// TIA Portal V17 export
// export: Created 2023-12-22T15:07:59.6202933Z, ExportSetting WithDefaults, DisplayName Totally Integrated Automation Portal, DisplayVersion V17, DisplayName TIA Portal Openness, DisplayVersion V17, DisplayName TIA Portal Version Control Interface, DisplayVersion V17, DisplayName STEP 7 Professional, DisplayVersion V17, DisplayName STEP 7 Safety, DisplayVersion V17, DisplayName WinCC Advanced, DisplayVersion V17
FUNCTION_BLOCK "PS_StartUp"   // FB13, LAD
{ S7_Optimized_Access := 'FALSE' }
VERSION : 0.1
// stored: AutoNumber false, IsIECCheckEnabled false, SetENOAutomatically false, UDAEnableTagReadback false
   VAR_INPUT
      PE : Real;
      LE_Target : Real;
      LE_Source : Real;
   END_VAR
   VAR_IN_OUT
      REQ : Int;
      Hz : Real;
   END_VAR
   VAR DB_SPECIFIC
      Start : Bool;   // Запуск системы
      Ready : Bool;   // Линия заполнена
      "Step" : Int;
      Warning : Word;
      PE_Point : Real;   // Давление на момент выхода плавный разгон
      PE_Delta : Real := 0.05;   // Допустимое отклонение
      PE_Min : Real;
      LE_Target_Point : Real;
      LE_Target_Delta : Real;
      LE_Target_Min : Real;
      LE_Source_Point : Real;
      LE_Source_Delta : Real;
      LE_Source_Min : Real;
      xSP : Array[0..5] of Struct
         Use { S7_SetPoint := 'True'} : Bool;
         REQ { S7_SetPoint := 'True'} : Int;
         Hz { S7_SetPoint := 'True'} : Real;
         PE { S7_SetPoint := 'True'} : Real;
         PE_Delta : Real;
      END_STRUCT;
   END_VAR
   VAR
      xTime { S7_SetPoint := 'True'} : Array[0..5] of "Time_M";
   END_VAR
   VAR_TEMP   // added for the SCL form of the ladder/FBD networks
      _w1 : Bool;
      _w2 : Bool;
      _w3 : Bool;
      _w4 : Bool;
      _w5 : Bool;
   END_VAR
BEGIN

REGION Network 1: 0 - Первичное заполнение труб
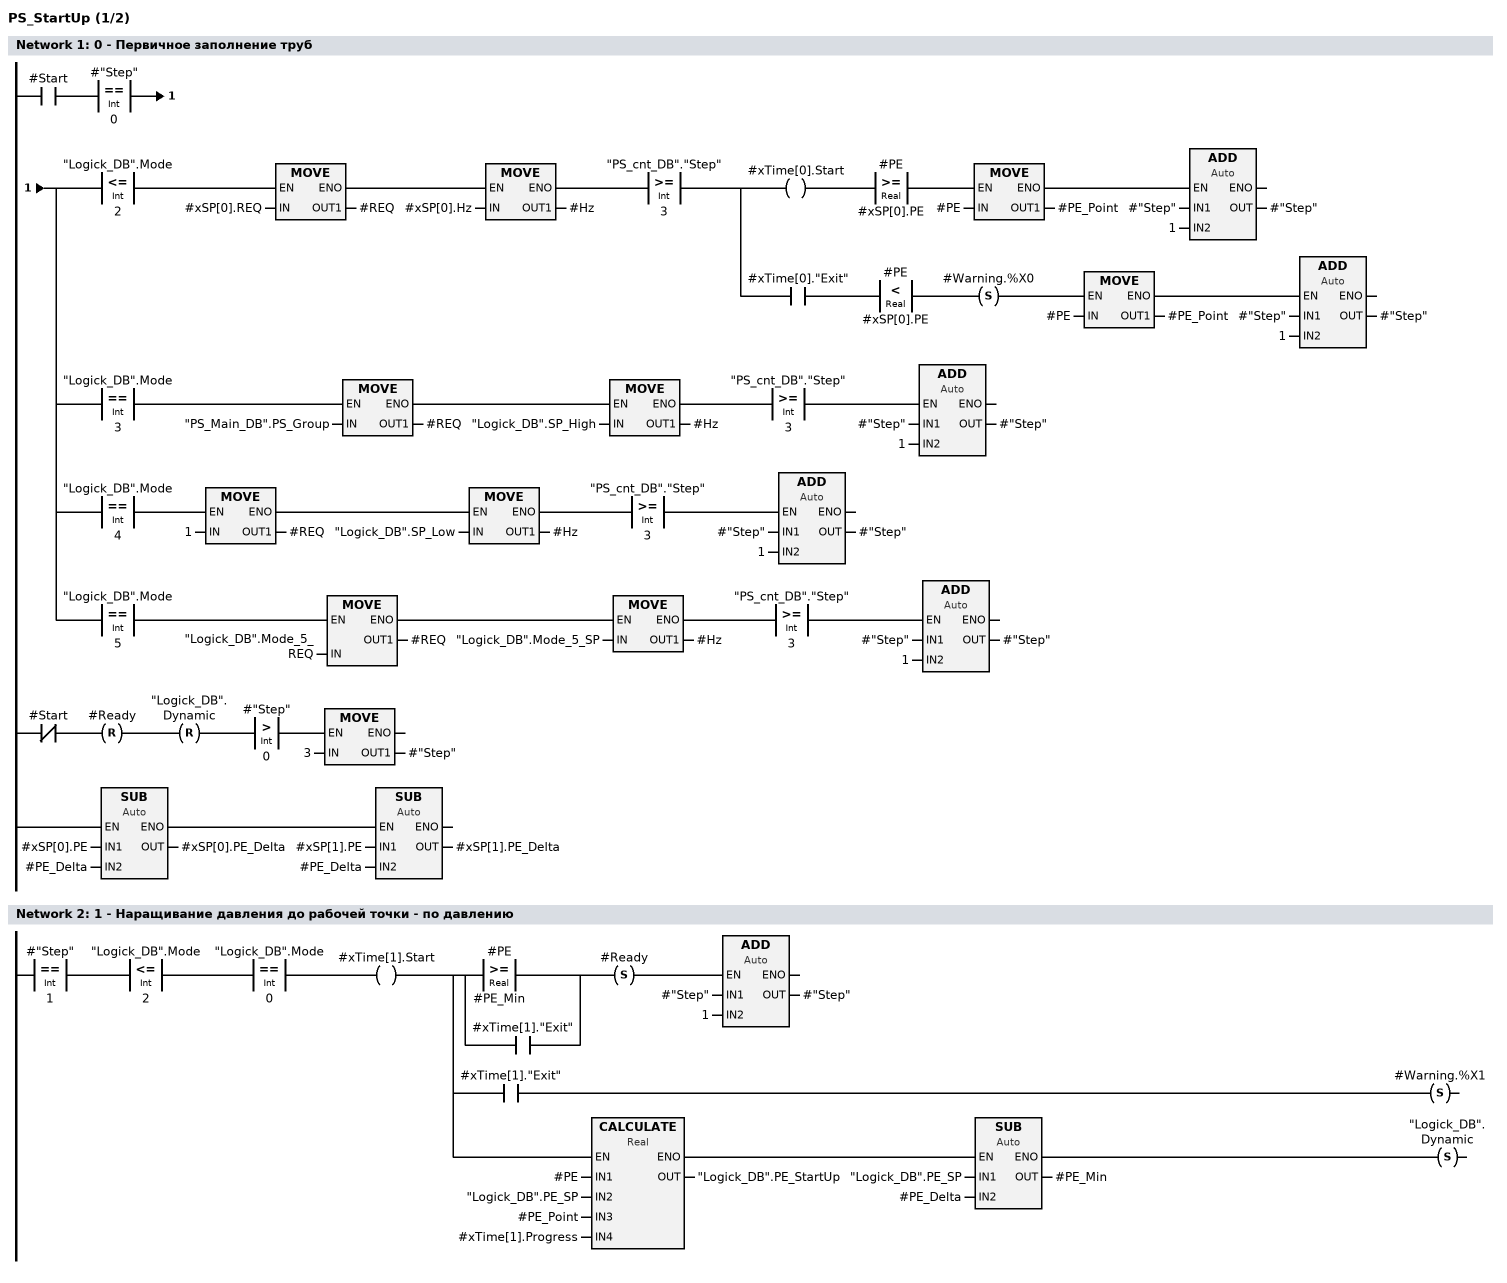
   RUNG wire#powerrail
      Contact( #Start )
      { S7_Templates := "SrcType := Int" } EQ_Contact(in1 := #"Step", in2 := 0)
      wire#w1
      { S7_Templates := "SrcType := Int" } LE_Contact(in1 := "Logick_DB".Mode, in2 := 2)
      Move(in := #xSP[0].REQ, out1 => #REQ)
      Move(in := #xSP[0].Hz, out1 => #Hz)
      { S7_Templates := "SrcType := Int" } GE_Contact(in1 := "PS_cnt_DB"."Step", in2 := 3)
      wire#w2
      Coil( #xTime[0].Start )
      { S7_Templates := "SrcType := Real" } GE_Contact(in1 := #PE, in2 := #xSP[0].PE)
      Move(in := #PE, out1 => #PE_Point)
      Add(in1 := #"Step", in2 := 1, out => #"Step")
   END_RUNG
   RUNG wire#w2
      Contact( #xTime[0]."Exit" )
      { S7_Templates := "SrcType := Real" } LT_Contact(in1 := #PE, in2 := #xSP[0].PE)
      S_Coil( #Warning.%X0 )
      Move(in := #PE, out1 => #PE_Point)
      Add(in1 := #"Step", in2 := 1, out => #"Step")
   END_RUNG
   RUNG wire#w1
      { S7_Templates := "SrcType := Int" } EQ_Contact(in1 := "Logick_DB".Mode, in2 := 3)
      Move(in := "PS_Main_DB".PS_Group, out1 => #REQ)
      Move(in := "Logick_DB".SP_High, out1 => #Hz)
      { S7_Templates := "SrcType := Int" } GE_Contact(in1 := "PS_cnt_DB"."Step", in2 := 3)
      Add(in1 := #"Step", in2 := 1, out => #"Step")
   END_RUNG
   RUNG wire#w1
      { S7_Templates := "SrcType := Int" } EQ_Contact(in1 := "Logick_DB".Mode, in2 := 4)
      Move(in := 1, out1 => #REQ)
      Move(in := "Logick_DB".SP_Low, out1 => #Hz)
      { S7_Templates := "SrcType := Int" } GE_Contact(in1 := "PS_cnt_DB"."Step", in2 := 3)
      Add(in1 := #"Step", in2 := 1, out => #"Step")
   END_RUNG
   RUNG wire#w1
      { S7_Templates := "SrcType := Int" } EQ_Contact(in1 := "Logick_DB".Mode, in2 := 5)
      Move(in := "Logick_DB".Mode_5_REQ, out1 => #REQ)
      Move(in := "Logick_DB".Mode_5_SP, out1 => #Hz)
      { S7_Templates := "SrcType := Int" } GE_Contact(in1 := "PS_cnt_DB"."Step", in2 := 3)
      Add(in1 := #"Step", in2 := 1, out => #"Step")
   END_RUNG
   RUNG wire#powerrail
      I_Contact( #Start )
      R_Coil( #Ready )
      R_Coil( "Logick_DB".Dynamic )
      { S7_Templates := "SrcType := Int" } GT_Contact(in1 := #"Step", in2 := 0)
      Move(in := 3, out1 => #"Step")
   END_RUNG
   RUNG wire#powerrail
      Sub(in1 := #xSP[0].PE, in2 := #PE_Delta, out => #xSP[0].PE_Delta)
      Sub(in1 := #xSP[1].PE, in2 := #PE_Delta, out => #xSP[1].PE_Delta)
   END_RUNG
   // the same network as SCL:
   #_w1 := #Start AND (#"Step" = 0);
   #_w2 := #_w1 AND ("Logick_DB".Mode <= 2);
   IF #_w2 THEN
       #REQ := #xSP[0].REQ;
       #Hz := #xSP[0].Hz;
   END_IF;
   #xTime[0].Start := #_w2 AND ("PS_cnt_DB"."Step" >= 3);
   IF #_w2 AND ("PS_cnt_DB"."Step" >= 3) AND (#PE >= #xSP[0].PE) THEN
       #PE_Point := #PE;
       #"Step" := #"Step" + 1;
   END_IF;
   IF #_w2 AND ("PS_cnt_DB"."Step" >= 3) AND #xTime[0]."Exit" AND (#PE < #xSP[0].PE) THEN
       #Warning.%X0 := TRUE;
       #PE_Point := #PE;
       #"Step" := #"Step" + 1;
   END_IF;
   #_w3 := #_w1 AND ("Logick_DB".Mode = 3);
   IF #_w3 THEN
       #REQ := "PS_Main_DB".PS_Group;
       #Hz := "Logick_DB".SP_High;
   END_IF;
   IF #_w3 AND ("PS_cnt_DB"."Step" >= 3) THEN #"Step" := #"Step" + 1; END_IF;
   #_w4 := #_w1 AND ("Logick_DB".Mode = 4);
   IF #_w4 THEN
       #REQ := 1;
       #Hz := "Logick_DB".SP_Low;
   END_IF;
   IF #_w4 AND ("PS_cnt_DB"."Step" >= 3) THEN #"Step" := #"Step" + 1; END_IF;
   #_w5 := #_w1 AND ("Logick_DB".Mode = 5);
   IF #_w5 THEN
       #REQ := "Logick_DB".Mode_5_REQ;
       #Hz := "Logick_DB".Mode_5_SP;
   END_IF;
   IF #_w5 AND ("PS_cnt_DB"."Step" >= 3) THEN #"Step" := #"Step" + 1; END_IF;
   IF NOT #Start THEN
       #Ready := FALSE;
       "Logick_DB".Dynamic := FALSE;
   END_IF;
   IF NOT #Start AND (#"Step" > 0) THEN #"Step" := 3; END_IF;
   #xSP[0].PE_Delta := #xSP[0].PE - #PE_Delta;
   #xSP[1].PE_Delta := #xSP[1].PE - #PE_Delta;
END_REGION

REGION Network 2: 1 - Наращивание давления до рабочей точки - по давлению
   RUNG wire#powerrail
      { S7_Templates := "SrcType := Int" } EQ_Contact(in1 := #"Step", in2 := 1)
      { S7_Templates := "SrcType := Int" } LE_Contact(in1 := "Logick_DB".Mode, in2 := 2)
      { S7_Templates := "SrcType := Int" } EQ_Contact(in1 := "Logick_DB".Mode, in2 := 0)
      Coil( #xTime[1].Start )
      wire#w1
      { S7_Templates := "SrcType := Real" } GE_Contact(in1 := #PE, in2 := #PE_Min)
      wire#w2
      S_Coil( #Ready )
      Add(in1 := #"Step", in2 := 1, out => #"Step")
   END_RUNG
   RUNG wire#w1
      Contact( #xTime[1]."Exit" )
   END_RUNG wire#w2
   RUNG wire#w1
      Contact( #xTime[1]."Exit" )
      S_Coil( #Warning.%X1 )
   END_RUNG
   RUNG wire#w1
      { S7_Templates := "SrcType := Real"; S7_Expression := "IN1 + (IN2 - IN3) * IN4" } Calculate(in1 := #PE, in2 := "Logick_DB".PE_SP, in3 := #PE_Point, in4 := #xTime[1].Progress, out => "Logick_DB".PE_StartUp)
      Sub(in1 := "Logick_DB".PE_SP, in2 := #PE_Delta, out => #PE_Min)
      S_Coil( "Logick_DB".Dynamic )
   END_RUNG
   // the same network as SCL:
   #xTime[1].Start := (#"Step" = 1) AND ("Logick_DB".Mode <= 2) AND ("Logick_DB".Mode = 0);
   #_w1 := (#"Step" = 1) AND ("Logick_DB".Mode <= 2) AND ("Logick_DB".Mode = 0);
   IF #_w1 AND ((#PE >= #PE_Min) OR #xTime[1]."Exit") THEN
       #Ready := TRUE;
       #"Step" := #"Step" + 1;
   END_IF;
   IF #_w1 AND #xTime[1]."Exit" THEN #Warning.%X1 := TRUE; END_IF;
   IF #_w1 THEN
       "Logick_DB".PE_StartUp := #PE + ("Logick_DB".PE_SP - #PE_Point) * #xTime[1].Progress;
       #PE_Min := "Logick_DB".PE_SP - #PE_Delta;
       "Logick_DB".Dynamic := TRUE;
   END_IF;
END_REGION

REGION Network 3: 1 - Наращивание давления до рабочей точки - по уровню в РЧВ
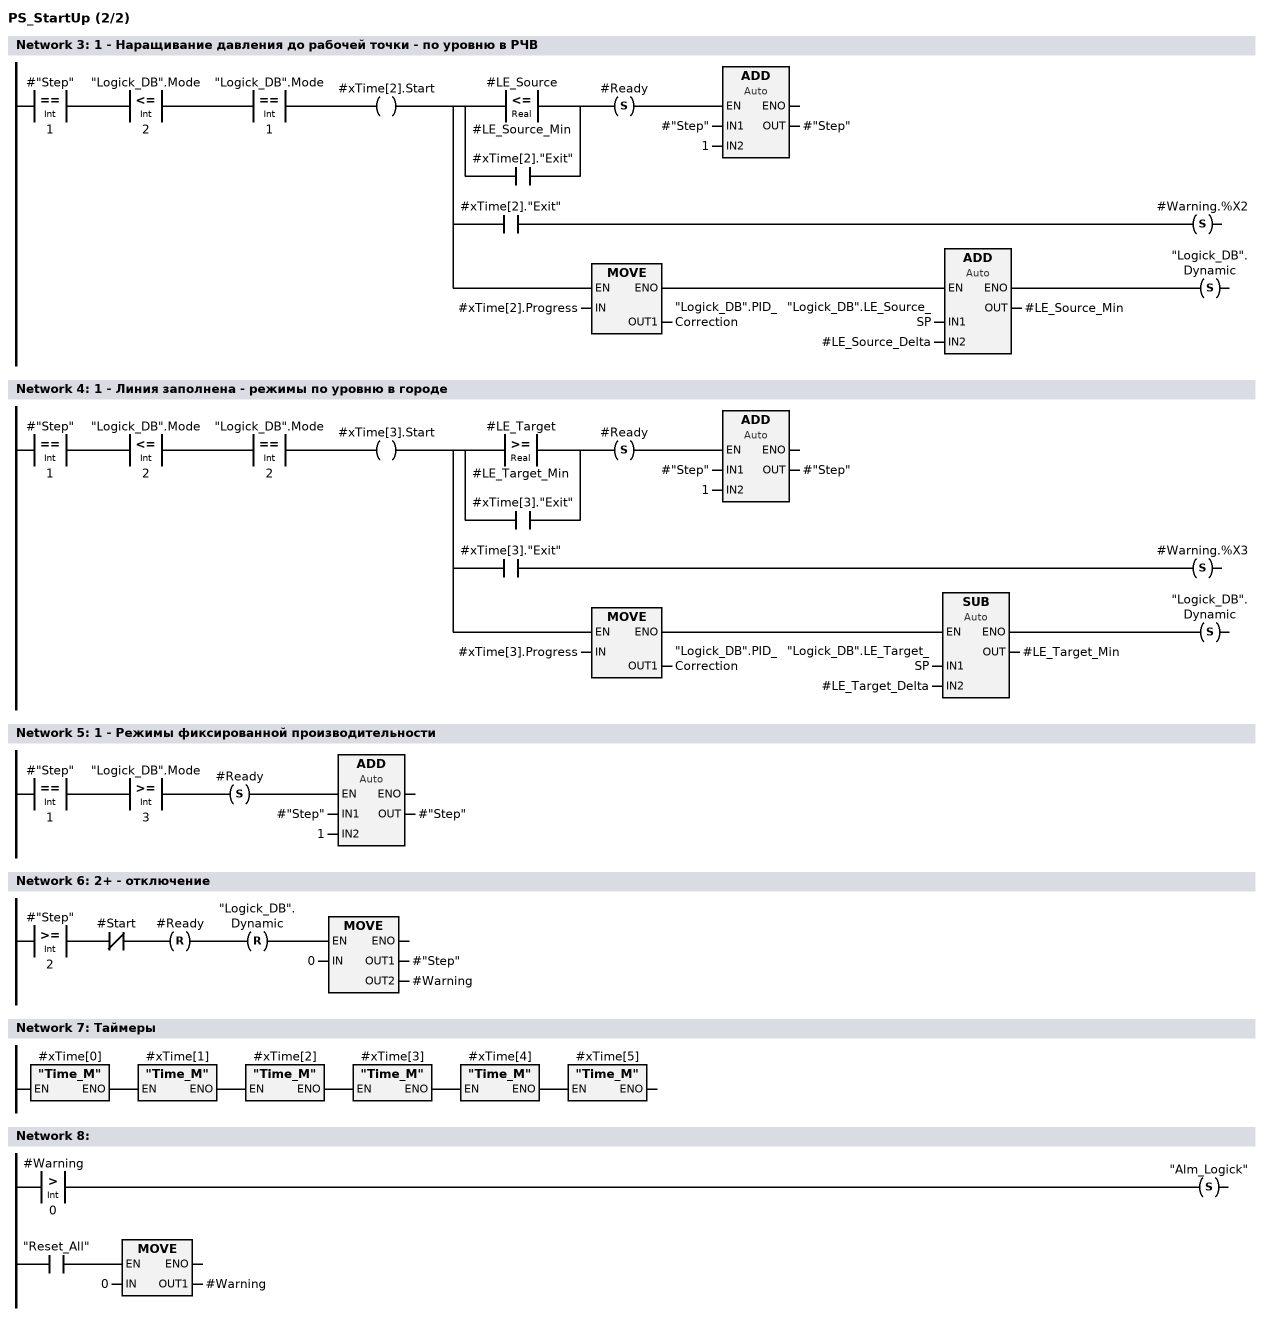
   RUNG wire#powerrail
      { S7_Templates := "SrcType := Int" } EQ_Contact(in1 := #"Step", in2 := 1)
      { S7_Templates := "SrcType := Int" } LE_Contact(in1 := "Logick_DB".Mode, in2 := 2)
      { S7_Templates := "SrcType := Int" } EQ_Contact(in1 := "Logick_DB".Mode, in2 := 1)
      Coil( #xTime[2].Start )
      wire#w1
      { S7_Templates := "SrcType := Real" } LE_Contact(in1 := #LE_Source, in2 := #LE_Source_Min)
      wire#w2
      S_Coil( #Ready )
      Add(in1 := #"Step", in2 := 1, out => #"Step")
   END_RUNG
   RUNG wire#w1
      Contact( #xTime[2]."Exit" )
   END_RUNG wire#w2
   RUNG wire#w1
      Contact( #xTime[2]."Exit" )
      S_Coil( #Warning.%X2 )
   END_RUNG
   RUNG wire#w1
      Move(in := #xTime[2].Progress, out1 => "Logick_DB".PID_Correction)
      Add(in1 := "Logick_DB".LE_Source_SP, in2 := #LE_Source_Delta, out => #LE_Source_Min)
      S_Coil( "Logick_DB".Dynamic )
   END_RUNG
   // the same network as SCL:
   #xTime[2].Start := (#"Step" = 1) AND ("Logick_DB".Mode <= 2) AND ("Logick_DB".Mode = 1);
   #_w1 := (#"Step" = 1) AND ("Logick_DB".Mode <= 2) AND ("Logick_DB".Mode = 1);
   IF #_w1 AND ((#LE_Source <= #LE_Source_Min) OR #xTime[2]."Exit") THEN
       #Ready := TRUE;
       #"Step" := #"Step" + 1;
   END_IF;
   IF #_w1 AND #xTime[2]."Exit" THEN #Warning.%X2 := TRUE; END_IF;
   IF #_w1 THEN
       "Logick_DB".PID_Correction := #xTime[2].Progress;
       #LE_Source_Min := "Logick_DB".LE_Source_SP + #LE_Source_Delta;
       "Logick_DB".Dynamic := TRUE;
   END_IF;
END_REGION

REGION Network 4: 1 - Линия заполнена - режимы по уровню в городе
   RUNG wire#powerrail
      { S7_Templates := "SrcType := Int" } EQ_Contact(in1 := #"Step", in2 := 1)
      { S7_Templates := "SrcType := Int" } LE_Contact(in1 := "Logick_DB".Mode, in2 := 2)
      { S7_Templates := "SrcType := Int" } EQ_Contact(in1 := "Logick_DB".Mode, in2 := 2)
      Coil( #xTime[3].Start )
      wire#w1
      { S7_Templates := "SrcType := Real" } GE_Contact(in1 := #LE_Target, in2 := #LE_Target_Min)
      wire#w2
      S_Coil( #Ready )
      Add(in1 := #"Step", in2 := 1, out => #"Step")
   END_RUNG
   RUNG wire#w1
      Contact( #xTime[3]."Exit" )
   END_RUNG wire#w2
   RUNG wire#w1
      Contact( #xTime[3]."Exit" )
      S_Coil( #Warning.%X3 )
   END_RUNG
   RUNG wire#w1
      Move(in := #xTime[3].Progress, out1 => "Logick_DB".PID_Correction)
      Sub(in1 := "Logick_DB".LE_Target_SP, in2 := #LE_Target_Delta, out => #LE_Target_Min)
      S_Coil( "Logick_DB".Dynamic )
   END_RUNG
   // the same network as SCL:
   #xTime[3].Start := (#"Step" = 1) AND ("Logick_DB".Mode <= 2) AND ("Logick_DB".Mode = 2);
   #_w1 := (#"Step" = 1) AND ("Logick_DB".Mode <= 2) AND ("Logick_DB".Mode = 2);
   IF #_w1 AND ((#LE_Target >= #LE_Target_Min) OR #xTime[3]."Exit") THEN
       #Ready := TRUE;
       #"Step" := #"Step" + 1;
   END_IF;
   IF #_w1 AND #xTime[3]."Exit" THEN #Warning.%X3 := TRUE; END_IF;
   IF #_w1 THEN
       "Logick_DB".PID_Correction := #xTime[3].Progress;
       #LE_Target_Min := "Logick_DB".LE_Target_SP - #LE_Target_Delta;
       "Logick_DB".Dynamic := TRUE;
   END_IF;
END_REGION

REGION Network 5: 1 - Режимы фиксированной производительности
   RUNG wire#powerrail
      { S7_Templates := "SrcType := Int" } EQ_Contact(in1 := #"Step", in2 := 1)
      { S7_Templates := "SrcType := Int" } GE_Contact(in1 := "Logick_DB".Mode, in2 := 3)
      S_Coil( #Ready )
      Add(in1 := #"Step", in2 := 1, out => #"Step")
   END_RUNG
   // the same network as SCL:
   IF (#"Step" = 1) AND ("Logick_DB".Mode >= 3) THEN
       #Ready := TRUE;
       #"Step" := #"Step" + 1;
   END_IF;
END_REGION

REGION Network 6: 2+ - отключение
   RUNG wire#powerrail
      { S7_Templates := "SrcType := Int" } GE_Contact(in1 := #"Step", in2 := 2)
      I_Contact( #Start )
      R_Coil( #Ready )
      R_Coil( "Logick_DB".Dynamic )
      Move(in := 0, out1 => #"Step", out2 => #Warning)
   END_RUNG
   // the same network as SCL:
   IF (#"Step" >= 2) AND NOT #Start THEN
       #Ready := FALSE;
       "Logick_DB".Dynamic := FALSE;
       #"Step" := 0;
       #Warning := 0;
   END_IF;
END_REGION

REGION Network 7: Таймеры
   RUNG wire#powerrail
      #xTime[0]()
      #xTime[1]()
      #xTime[2]()
      #xTime[3]()
      #xTime[4]()
      #xTime[5]()
   END_RUNG
   // the same network as SCL:
   #xTime[0](ENO => #_w1);   // "Time_M"
   #xTime[1](EN := #_w1, ENO => #_w2);   // "Time_M"
   #xTime[2](EN := #_w2, ENO => #_w3);   // "Time_M"
   #xTime[3](EN := #_w3, ENO => #_w4);   // "Time_M"
   #xTime[4](EN := #_w4, ENO => #_w5);   // "Time_M"
   IF #_w5 THEN
       #xTime[5]();   // "Time_M"
   END_IF;
END_REGION

REGION Network 8
   RUNG wire#powerrail
      { S7_Templates := "SrcType := Int" } GT_Contact(in1 := #Warning, in2 := 0)
      S_Coil( "Alm_Logick" )
   END_RUNG
   RUNG wire#powerrail
      Contact( "Reset_All" )
      Move(in := 0, out1 => #Warning)
   END_RUNG
   // the same network as SCL:
   IF #Warning > 0 THEN "Alm_Logick" := TRUE; END_IF;
   IF "Reset_All" THEN #Warning := 0; END_IF;
END_REGION
END_FUNCTION_BLOCK
